(* IEC 61131-3 sources: HMITools/, 11 files *)

(* ---- GetDataObjectList.st ---- *)
(*  *)
FUNCTION GetDataObjectList

		//Keep track of the objects that we've gone through
	//unsigned int objectIndex = 0;
	objectIndex:= 0;

	//Number of variables that have been found
	numberVariables:=0;
	duplicate:=0;
	index:=0;

	//Check for valid inputs
	IF( List = 0 ) THEN
		GetDataObjectList:=0;
		RETURN;
	END_IF

	//Clear out any bad data
	Files ACCESS List;
	brsmemset(ADR(Files ),0,MaxObjects*(LIST_BOX_STRING_SIZE+1));

	//Look through all the objects
	WHILE( MO_list(objectIndex, ADR(objectIndex), ADR(Item)) = 0 AND numberVariables < MaxObjects)DO
		//If it is a cyclic object check if it has the variable
		duplicate:=0;
		IF( Item.type = 16#41) THEN
			FOR index:= 0 TO numberVariables DO
				IF(brsstrcmp(ADR(Item.name),ADR(Files[index]))=0)THEN
					duplicate:=1;
					EXIT;
				END_IF
			END_FOR
			IF(NOT duplicate) THEN
				brsstrcpy( ADR(Files[numberVariables]),ADR(Item.name));
				numberVariables:=numberVariables+1;
			END_IF
		END_IF
	END_WHILE

	//Return the number of found variables to make it easy to add to the list outside the function.
	GetDataObjectList:= numberVariables;

END_FUNCTION

(* ---- HMI_Lock.st ---- *)
(********************************************************************
 * COPYRIGHT --
 ********************************************************************
 * Library: HMI_Basic
 * File: HMI_Lock.st
 * Author: David
 * Created: May 03, 2011
 ********************************************************************
 * Implementation of library HMI_Basic
 ********************************************************************)

(****************************************************************)
(* Lock an item on the screen 									*)
(****************************************************************)

(* Function			DONE and TESTED DFB 20110503 *)

FUNCTION HMI_Lock

(****************************************************************)
(* Set return value to get rid of compiler error				*)
(****************************************************************)

HMI_Lock:=	FALSE;

(****************************************************************)
(* Set/clear proper bit in StatusDP								*)
(****************************************************************)

StatusDP.HMI_STATBIT_LOCK:=	HMI_LOCKED;

END_FUNCTION

(* ---- HMI_OpenTouchpad.st ---- *)
(********************************************************************
 * COPYRIGHT --
 ********************************************************************
 * Library: HMI_Basic
 * File: HMI_OpenTouchpad.st
 * Author: David
 * Created: May 04, 2011
 ********************************************************************
 * Implementation of library HMI_Basic
 ********************************************************************)

(********************************************************************)
(* Opens the touchpad for an item on the screen 					*)
(********************************************************************)

(* Function			DONE and TESTED DFB 20110504 *)

FUNCTION HMI_OpenTouchpad

(****************************************************************)
(* Set return value to get rid of compiler error				*)
(****************************************************************)

HMI_OpenTouchpad:=	FALSE;

(****************************************************************)
(* Set/clear proper bit in StatusDP								*)
(****************************************************************)

StatusDP.HMI_STATBIT_TOUCHPAD:=	1;

END_FUNCTION

(* ---- HMI_ResetFocus.st ---- *)
(********************************************************************
 * COPYRIGHT --
 ********************************************************************
 * Library: HMI_Basic
 * File: HMI_ResetFocus.st
 * Author: David
 * Created: May 04, 2011
 ********************************************************************
 * Implementation of library HMI_Basic
 ********************************************************************)

(************************************************************************************)
(* Resets the focus bit for an item on the screen. THIS DOES NOT MOVE THE FOCUS!	*)
(************************************************************************************)

(* Function			DONE and TESTED DFB 20110504 *)

FUNCTION HMI_ResetFocus

(****************************************************************)
(* Set return value to get rid of compiler error				*)
(****************************************************************)

HMI_ResetFocus:=	FALSE;

(****************************************************************)
(* Set/clear proper bit in StatusDP								*)
(****************************************************************)

StatusDP.HMI_STATBIT_FOCUS:=	0;

END_FUNCTION

(* ---- HMI_SetFocus.st ---- *)
(********************************************************************
 * COPYRIGHT --
 ********************************************************************
 * Library: HMI_Basic
 * File: HMI_SetFocus.st
 * Author: David
 * Created: May 04, 2011
 ********************************************************************
 * Implementation of library HMI_Basic
 ********************************************************************)

(********************************************************************)
(* Sets the focus for an item on the screen. FOCUS MUST BE RESET!	*)
(********************************************************************)

(* Function			DONE and TESTED DFB 20110504 *)

FUNCTION HMI_SetFocus

(****************************************************************)
(* Set return value to get rid of compiler error				*)
(****************************************************************)

HMI_SetFocus:=	FALSE;

(****************************************************************)
(* Set/clear proper bit in StatusDP								*)
(****************************************************************)

StatusDP.HMI_STATBIT_FOCUS:=	1;

END_FUNCTION

(* ---- HMI_Show.st ---- *)
(********************************************************************
 * COPYRIGHT --
 ********************************************************************
 * Library: HMI_Basic
 * File: HMI_Show.st
 * Author: David
 * Created: May 03, 2011
 ********************************************************************
 * Implementation of library HMI_Basic
 ********************************************************************)

(****************************************************************)
(* Show an item on the screen 									*)
(****************************************************************)

(* Function			DONE and TESTED DFB 20110503 *)

FUNCTION HMI_Show

(****************************************************************)
(* Set return value to get rid of compiler error				*)
(****************************************************************)

HMI_Show:=	FALSE;

(****************************************************************)
(* Set/clear proper bit in StatusDP								*)
(****************************************************************)

StatusDP.HMI_STATBIT_VIS:=	HMI_VISIBLE;

END_FUNCTION

(* ---- HMI_Unlock.st ---- *)
(********************************************************************
 * COPYRIGHT --
 ********************************************************************
 * Library: HMI_Basic
 * File: HMI_Unlock.st
 * Author: David
 * Created: May 03, 2011
 ********************************************************************
 * Implementation of library HMI_Basic
 ********************************************************************)

(****************************************************************)
(* Unlock an item on the screen 								*)
(****************************************************************)

(* Function			DONE and TESTED DFB 20110503 *)

FUNCTION HMI_Unlock

(****************************************************************)
(* Set return value to get rid of compiler error				*)
(****************************************************************)

HMI_Unlock:=	FALSE;

(****************************************************************)
(* Set/clear proper bit in StatusDP								*)
(****************************************************************)

StatusDP.HMI_STATBIT_LOCK:=	HMI_UNLOCKED;

END_FUNCTION

(* ---- DirectoryFub.st ---- *)
(********************************************************************
 * COPYRIGHT -- Automation Resources Group
 ********************************************************************
 * Program: FileManager
 * File: Directory.st
 * Author: Josh
 * Created: April 01, 2012
 ********************************************************************
 * Implementation of program FileManager
 ********************************************************************)

(*  *)
FUNCTION_BLOCK DirectoryFub

IF FileList = 0 OR Enable = 0 THEN
	Updating:=0;
	RETURN;
END_IF

Files ACCESS FileList;

	// Step through all states faster by looping 5 times
	FOR index:=0 TO 5 DO

		CASE State OF
			0:
				DirectoryRead.enable:=0;
				//CurrentFileIndex:=0; This variable is never used again.
				Updating:=1;
				State:=1;

			1:
				DirectoryOpen.enable := 	TRUE;
				DirectoryOpen.pDevice := 	ADR(FileDevice);
				DirectoryOpen.pName := 		pPath;
				DirectoryOpen();
				IF DirectoryOpen.status < ERR_FUB_ENABLE_FALSE THEN
					IF DirectoryOpen.status = ERR_OK THEN
						Ident :=			DirectoryOpen.ident;
						DirectoryOpen.enable:=	 FALSE;
						State:= 			State+1;
					ELSE
						status:= 			DirectoryOpen.status;
						State:=				10;
					END_IF;
				ELSE
					EXIT;
				END_IF;
				brsmemset(ADR(Files),0,MaxValues*(LIST_BOX_STRING_SIZE+1));
				ListFileIndex:=		0;
				status:=			ERR_FUB_BUSY;

			2:
				//read directory
				DirectoryRead.enable := 	TRUE;
				DirectoryRead.ident := 		Ident;
				DirectoryRead.pData := 		ADR(DirData);
				DirectoryRead.data_len := 	SIZEOF(DirData);
				DirectoryRead();
				IF DirectoryRead.status < ERR_FUB_ENABLE_FALSE THEN
					IF DirectoryRead.status = ERR_OK THEN
						DirectoryRead.enable := FALSE;
						State:= 			State+1;
					ELSIF DirectoryRead.status = fiERR_NO_MORE_ENTRIES THEN
						NumFiles:= 			ListFileIndex;
						status:=			ERR_OK;
						State:=				5;
					ELSE
						IF DirectoryRead.status = 20799 THEN
							status:= FileIoGetSysError();
						ELSE
							status:= DirectoryRead.status;
						END_IF;
						State:=				10;
					END_IF;
				ELSE
					EXIT;
				END_IF;

			3:
				brsstrcpy(ADR(TempString),ADR(DirData.Filename));
				iNameFilter:=NameFilter;
				//If file extension filter defined
				IF FileExt <> '' THEN
					brsmemset(ADR(TempExtension),0,SIZEOF(TempExtension));
					TempExtension:=	'.';
					brsstrcat(ADR(TempExtension),ADR(FileExt));
					//item is a File, files are filtered
					IF DirData.Mode = fiFILE THEN
						//compare just the selected extension from the file name + extension (e.g. compare ".csv" from "testing.csv")
						IF ( brsmemcmp((ADR(TempString)+(brsstrlen(ADR(TempString))-(brsstrlen(ADR(TempExtension)))))
							, ADR(TempExtension)
							, brsstrlen(ADR(TempExtension))) = 0) THEN

							//convert NameFilter to lowercase
							brsmemset(ADR(lcNameFilter),0,SIZEOF(lcNameFilter));
							FOR i:= 0 TO (SIZEOF(NameFilter) - 1) DO
								brsmemcpy(ADR(IsolatedChar),(ADR(NameFilter) + i),SIZEOF(USINT));
								IF IsolatedChar = 0 THEN// OR IsolatedChar = 46 THEN//if null or '.', dont convert file extension to lc
									EXIT;
								ELSIF IsolatedChar >=  65 AND IsolatedChar <=  90  THEN//Uppser case ascii
									brsmemset((ADR(lcNameFilter) + i),(IsolatedChar + 32),SIZEOF(USINT));
								ELSE//lower case ascii
									brsmemset((ADR(lcNameFilter) + i),IsolatedChar,SIZEOF(USINT));
								END_IF;
							END_FOR;
							//convert TempString to lowercase
							brsmemset(ADR(lcTempString),0,SIZEOF(lcTempString));
							FOR i:= 0 TO (SIZEOF(TempString) - 1) DO
								brsmemcpy(ADR(IsolatedChar),(ADR(TempString) + i),SIZEOF(USINT));
								IF IsolatedChar = 0 THEN// OR IsolatedChar = 46 THEN//if null or '.', dont convert file extension to lc
									EXIT;
								ELSIF IsolatedChar >=  65 AND IsolatedChar <=  90  THEN//Uppser case ascii
									brsmemset((ADR(lcTempString) + i),(IsolatedChar + 32),SIZEOF(USINT));
								ELSE//lower case ascii
									brsmemset((ADR(lcTempString) + i),IsolatedChar,SIZEOF(USINT));
								END_IF;
							END_FOR;
							brsmemcpy(ADR(IsolatedChar),ADR(TempString),SIZEOF(USINT));

							//Compare both lower case strings
							//Check for hidden files
							IF (FIND(lcTempString, lcNameFilter) <> 0) AND (ShowHiddenFiles OR IsolatedChar <> 46) THEN
								brsstrcpy(ADR(Files[ListFileIndex]),ADR(DirData.Filename));
								ListFileIndex:=		ListFileIndex+1;
								State:= 			State+1;
							ELSE
								State:= 			State+1;
							END_IF;

						ELSE
							State:= 			State+1;
						END_IF
					//item is a Directory, directories are not filtered
					ELSIF EnableDirectorySearch AND (brsstrcmp(ADR(DirData.Filename),ADR('.')) <> 0) THEN
						IF ((brsstrcmp(pPath,ADR('')) = 0) AND ((brsstrcmp(ADR(DirData.Filename),ADR('..')) = 0))) THEN
							State:=				State+1;
						ELSE
							brsstrcpy(ADR(Files[ListFileIndex]),ADR('\'));
							brsstrcat(ADR(Files[ListFileIndex]),ADR(DirData.Filename));
							ListFileIndex:=		ListFileIndex+1;
							State:=				State+1;
						END_IF;
					ELSE//if a directory and enabledirectorysearch is false
						State:= 				State+1;
					END_IF;
				//No extension filter defined
				ELSE
					//item is a File, files are filtered
					IF DirData.Mode = fiFILE THEN
						//convert NameFilter to lowercase
						brsmemset(ADR(lcNameFilter),0,SIZEOF(lcNameFilter));
						FOR i:= 0 TO (SIZEOF(NameFilter) - 1) DO
							brsmemcpy(ADR(IsolatedChar),(ADR(NameFilter) + i),SIZEOF(USINT));
							IF IsolatedChar = 0 THEN// OR IsolatedChar = 46 THEN//if null or '.', dont convert file extension to lc
								EXIT;
							ELSIF IsolatedChar >=  65 AND IsolatedChar <=  90  THEN//Uppser case ascii
								brsmemset((ADR(lcNameFilter) + i),(IsolatedChar + 32),SIZEOF(USINT));
							ELSE//lower case ascii
								brsmemset((ADR(lcNameFilter) + i),IsolatedChar,SIZEOF(USINT));
							END_IF;
						END_FOR;
						//convert TempString to lowercase
						brsmemset(ADR(lcTempString),0,SIZEOF(lcTempString));
						FOR i:= 0 TO (SIZEOF(TempString) - 1) DO
							brsmemcpy(ADR(IsolatedChar),(ADR(TempString) + i),SIZEOF(USINT));
							IF IsolatedChar = 0 THEN//OR IsolatedChar = 46 THEN//if null or '.', dont convert file extension to lc
								EXIT;
							ELSIF IsolatedChar >=  65 AND IsolatedChar <=  90  THEN//Uppser case ascii
								brsmemset((ADR(lcTempString) + i),(IsolatedChar + 32),SIZEOF(USINT));
							ELSE//lower case ascii
								brsmemset((ADR(lcTempString) + i),IsolatedChar,SIZEOF(USINT));
							END_IF;
						END_FOR;

						brsmemcpy(ADR(IsolatedChar),ADR(TempString),SIZEOF(USINT));

						//Compare both lower case strings
						//Check for hidden files
						IF (FIND(lcTempString, lcNameFilter) <> 0) AND (ShowHiddenFiles OR IsolatedChar <> 46) THEN
							brsstrcpy(ADR(Files[ListFileIndex]),ADR(DirData.Filename));
							ListFileIndex:=		ListFileIndex+1;
							State:= 			State+1;
						ELSE
							State:= 			State+1;
						END_IF;

					//item is a Directory, directories are not filtered
					ELSIF EnableDirectorySearch AND (brsstrcmp(ADR(DirData.Filename),ADR('.')) <> 0) THEN //item is a Directory, directories are not filtered
						IF ((brsstrcmp(pPath,ADR('')) = 0) AND ((brsstrcmp(ADR(DirData.Filename),ADR('..')) = 0))) THEN
							State:=				State+1;
						ELSE
							brsstrcpy(ADR(Files[ListFileIndex]),ADR('\'));
							brsstrcat(ADR(Files[ListFileIndex]),ADR(DirData.Filename));
							ListFileIndex:=		ListFileIndex+1;
							State:=				State+1;
						END_IF;
					ELSE//if a directory and enabledirectorysearch is false
						State:= 				State+1;
					END_IF;
				END_IF;

			4:
				IF ListFileIndex = MaxValues THEN
					status:=	ERR_OK;
					NumFiles:= 	ListFileIndex;
					State:=		5;
				ELSE
					State:=		2;
				END_IF;

			5:
				DirectoryClose.enable := 	TRUE;
				DirectoryClose.ident := 	Ident;
				DirectoryClose();
				IF DirectoryClose.status = ERR_OK THEN
					DirectoryClose.enable := FALSE;
					State:= 				6;
				END_IF;

			10:
				Initialized:=	1;
				UpdateTimer.IN:=1;
				IF UpdateTimer.Q OR iNameFilter<>NameFilter OR Refresh THEN
					Refresh:= 	0;
					State:=		0;
				END_IF

			ELSE
				Initialized:=	1;
				Updating:=		0;
				UpdateTimer.IN:=1;
				IF UpdateTimer.Q OR iNameFilter<>NameFilter OR Refresh THEN
					Refresh:= 	0;
					State:=		0;
				END_IF
		END_CASE;
	END_FOR;

UpdateTimer.PT:=T#60s;
UpdateTimer();
UpdateTimer.IN:=0;

END_FUNCTION_BLOCK

(* ---- HMI_File_Browse.st ---- *)
(********************************************************************
 * COPYRIGHT --
 ********************************************************************
 * Library: HMITools
 * File: HMIFileBrowse.st
 * Author: Josh
 * Created: November 08, 2012
 ********************************************************************
 * Implementation of library HMITools
 ********************************************************************)

FUNCTION_BLOCK HMIFileBrowse
	// Error Checks

	IF pFileList = 0 THEN
		Status :=	'Invalid entry: FileList = 0';
		RETURN;
	END_IF;

	IF MaxFiles = 0 THEN
		Status :=	'Invalid entry: MaxFiles = 0';
		RETURN;
	END_IF;

	IF pFileExtList = 0
		AND MaxExt <> 0 THEN
		Status :=	'Invalid entry: pFileExtList = 0';
		RETURN;
	END_IF;

	IF pFileExtList <> 0
		AND MaxExt = 0 THEN
		Status :=	'Invalid entry: MaxExt = 0';
		RETURN;
	END_IF;

	IF FileDevice = '' THEN
		Status :=	'Invalid entry: FileDevice = 0';
		RETURN;
	END_IF;

	IF BrowseToDirectory AND EnableDirectorySearch = FALSE THEN
		BrowseToDirectory:=	FALSE;
		Status :=	'Please enable directory search';
	END_IF;

	IF Internal.TempFileList = 0 THEN
		TMP_alloc(SIZEOF(FileSelection) * MaxFiles ,ADR(Internal.TempFileList));
	END_IF

	Internal.FileExtensionSelector.IndexDP:=FileExtIndex;
	Internal.FileExtensionSelector.Enable:=Enable;
	Internal.FileExtensionSelector.MaxDP:=MaxExt;
	Internal.FileExtensionSelector.Selection:=ADR(FileExtSelection);
	IF pFileExtList <> 0 THEN
		Internal.FileExtensionSelector.SelectionList:=pFileExtList;
	END_IF;
	Internal.FileExtensionSelector();

	Internal.Directory.Enable:=		Enable AND NOT EnableDataObjects;
	Internal.Directory.MaxValues:= 	MaxFiles;
	IF Internal.TempFileList <> 0 THEN
		Internal.Directory.FileList:=Internal.TempFileList;
	ELSE
		Internal.Directory.FileList:=pFileList;
	END_IF

	//If initial path given
	IF pDirectorySearchPath <> 0
		AND Internal.InternalBrowsingPath = '' THEN
		brsstrcpy(ADR(CurrentPath),pDirectorySearchPath);
	END_IF;

	//if command to add FileSelection to browsing path,
	IF BrowseToDirectory
		AND FileSelection <> '\..'
		AND FileSelection <> '' THEN
		BrowseToDirectory := 	FALSE;
		Refresh := 1; // do an update and navigate to directory

		//Running directory path check
		brsmemcpy(ADR(Internal.IsolatedChar),ADR(FileSelection),SIZEOF(USINT));
		IF Internal.IsolatedChar = ASCII_BACKSLASH THEN
			//add selected file to internal path
			brsstrcat(ADR(Internal.InternalBrowsingPath),(ADR(FileSelection) + 1));//Don't add first character "\" to the browsing path
			brsstrcat(ADR(Internal.InternalBrowsingPath),ADR('\'));
			//reset current path
			brsmemset(ADR(CurrentPath),0,SIZEOF(CurrentPath));
			//repopulate current path with directory path input
			IF pDirectorySearchPath <> 0 THEN
				brsstrcpy(ADR(CurrentPath),(pDirectorySearchPath));
			END_IF;
			brsstrcat(ADR(CurrentPath),ADR(Internal.InternalBrowsingPath));
			//RESET FileSelection
			FileIndex:=				-1;
			FileSelection:=			'';
		ELSE
			Status:= 				'Invalid Internal.Directory';
		END_IF;
	//If command GoToParentInternal.Directory
	ELSIF BrowseToDirectory AND FileSelection = '\..' THEN
		BrowseToDirectory :=	FALSE;
		Refresh := 1; // do an update and navigate to directory
		Internal.PathStrSize:=		UDINT_TO_UINT(brsstrlen(ADR(Internal.InternalBrowsingPath)));
		IF Internal.InternalBrowsingPath = '' THEN//at highest allowed directory, indicated by input FileDevice and Path
			Status:= 				'Invalid Internal.Directory';
		ELSE
			brsmemset(ADR(Internal.InternalBrowsingPath) +(Internal.PathStrSize - 1 ),0,SIZEOF(USINT));//remove the last character "\"
			FOR Internal.i:= 1 TO Internal.PathStrSize DO
				//isolate a single character off of the path string
				brsmemcpy(ADR(Internal.IsolatedChar),ADR(Internal.InternalBrowsingPath)+(Internal.PathStrSize-Internal.i),SIZEOF(USINT));
				//if no characters left
				IF brsstrcmp(ADR(Internal.InternalBrowsingPath),ADR('')) = 0 THEN
					EXIT;
				//if found a backslash character at the end of the string, remove it and exit
				ELSIF Internal.IsolatedChar = ASCII_BACKSLASH  THEN
					EXIT;
				//else it's a normal character, remove it
				ELSE
					brsmemset(ADR(Internal.InternalBrowsingPath) +(Internal.PathStrSize-Internal.i),0,SIZEOF(USINT));
				END_IF;
			END_FOR;
		END_IF;
		//RESET FileSelection
		FileIndex:=		-1;
		FileSelection:=	'';
		//set output to current path
		brsmemset(ADR(CurrentPath),0,SIZEOF(CurrentPath));
		IF pDirectorySearchPath <> 0 THEN
			brsstrcpy(ADR(CurrentPath),pDirectorySearchPath);
		END_IF;
		brsstrcat(ADR(CurrentPath),ADR(Internal.InternalBrowsingPath));
	ELSIF BrowseToDirectory AND FileSelection = '' THEN
		BrowseToDirectory :=	FALSE;
		Status :=	'Invalid Internal.Directory';
	END_IF;

	//If selecting a file from listbox don't update name filter
	IF FileIndex < 0 THEN
		Internal.NameFilter :=	FileSelection;
	END_IF

	//temporarly display the filter being applied
	IF FileIndex < 0 AND Internal.NameFilter <> '' THEN
		Status :=		'Filter "';
		brsstrcat(ADR(Status),ADR(Internal.NameFilter));
		brsstrcat(ADR(Status),ADR('" applied'));
	END_IF

	//Reset Internal.NameFilter if a space character is the first character
	IF (brsmemcmp(ADR(FileSelection),ADR(' '),1) = 0) THEN
		Internal.NameFilter:=		'';
		FileSelection :=	'';
		Status :=			'Name filter removed';
	END_IF

	Internal.Directory.FileExt:=		FileExtSelection;
	Internal.Directory.FileDevice:=		FileDevice;
	Internal.Directory.EnableDirectorySearch:=	EnableDirectorySearch;
	Internal.Directory.pPath:=			ADR(CurrentPath);
	Internal.Directory.NameFilter:= 	Internal.NameFilter;

	IF (Refresh) THEN
		Internal.Directory.Refresh := 1;
	END_IF

	Internal.Directory();
	Refresh := 0;

	IF EnableDataObjects AND Enable THEN
		NumFiles:= GetDataObjectList(Internal.Directory.FileList,MaxFiles);
	ELSE
		NumFiles:= 				Internal.Directory.NumFiles;
	END_IF

	IF NOT Internal.Directory.Updating
		AND Internal.TempFileList <> 0
		AND Enable
		THEN
		brsmemcpy(pFileList,Internal.TempFileList,Internal.Directory.MaxValues*(LIST_BOX_STRING_SIZE+1));
	END_IF

	//If manually changing FileSelection, reset with FileIndex to update the Internal.NameFilter
	IF Internal.oldFileSelection <> FileSelection AND FileIndex = Internal.oldFileIndex THEN
		FileIndex:=	-1;
	END_IF;

	Internal.TempFileSelection := FileSelection;

	Internal.FileNameSelector.IndexDP:=		FileIndex;
	Internal.FileNameSelector.Enable:=		Enable;
	Internal.FileNameSelector.Enable:=		TRUE;
	Internal.FileNameSelector.MaxDP:=		Internal.Directory.NumFiles;
	Internal.FileNameSelector.Selection:=	ADR(Internal.TempFileSelection);
	Internal.FileNameSelector.SelectionList:=	pFileList;
	Internal.FileNameSelector();

	//We need to read back the found index to ensure that we aren't constantly updating
	FileIndex:= Internal.FileNameSelector.IndexDP;

	FileExtIndex:=	Internal.FileExtensionSelector.IndexDP;
	//FileIndex:=Internal.oldFileSelection.IndexDP;

	IF FileIndex > -1 THEN
		FileSelection:=		Internal.TempFileSelection;
		Internal.oldFileSelection:=	FileSelection;
	END_IF;

	CompletionDP:=Internal.FileNameSelector.CompletionDP;

	//If manually changing FileSelection, reset with FileIndex to update the Internal.NameFilter
	IF Internal.oldFileSelection <> FileSelection AND FileIndex = Internal.oldFileIndex THEN
		FileIndex:=	-1;
		Internal.oldFileSelection:=	FileSelection;
	ELSE
		Internal.oldFileSelection:=	FileSelection;
	END_IF;
	IF Internal.oldFileIndex <> FileIndex THEN
		Internal.oldFileIndex:=		FileIndex;
	END_IF;

	//Reset Error String Handling
	IF Status <> '' THEN
		Internal.TON_0.IN := 	TRUE;
		Internal.TON_0.PT := 	T#2s;
		IF Internal.TON_0.Q THEN
			Internal.TON_0.IN:=	FALSE;
			brsmemset(ADR(Status),0,SIZEOF(Status));
		END_IF;
	ELSE
		Internal.TON_0.IN := 	FALSE;
	END_IF;
	Internal.TON_0();

	//If no files or directories found
	IF NumFiles = 0 AND EnableDirectorySearch = FALSE THEN
		Status:=	'No files found';
	ELSIF NumFiles = 0 AND EnableDirectorySearch = TRUE THEN
		Status:=	'No items found';
	END_IF;

END_FUNCTION_BLOCK

(* ---- Trend_ZoomScroll.st ---- *)
(********************************************************************
 * COPYRIGHT -- Automation Resources Group
 ********************************************************************
 * Library: HMITools
 * File: Trend_ZoomScroll.st
 * Author: David
 * Created: October 25, 2010
 ********************************************************************
 * Implementation of library HMITools
 ********************************************************************)

(********************************************************************)
(* Smart handling of trend zooming and scaling 						*)
(********************************************************************)

(* Functionality			DONE and TESTED DFB *)

FUNCTION_BLOCK Trend_ZoomScroll

	(* Initialize values on startup *)

	IF( NOT(Init) )THEN

 		Init:=	1;
		Reset:=	1;

	END_IF

	(* Reset *)

	IF( Reset )THEN

 		Reset:=		0;

		ZoomDP:=	1;
		ScrollDP:=	0;
		ModeDP:=	1;

	END_IF

	(* Zoom *)

	(* Check ZoomBase *)

	IF( ZoomBase < 1 )THEN

		(* If ZoomBase is less than 1, this will cause problems.
			Default to a ZoomBase of 1. This cancels out all Zooming *)

 		ZoomBase:=	1;

	END_IF

	IF( ZoomIn )THEN

 		ZoomIn:=	0;

		Midpt:=		ScrollDP + (0.5 / ZoomDP);	(* Midpt is ScrollDP (StartPt_curr) + Range_curr/2; Range_curr is 1/ZoomDP_curr *)
		ZoomDP:=	ZoomDP * ZoomBase; 			(* Zoom is increased by ZoomBase *)
		ScrollDP:=	Midpt - (0.5 / ZoomDP);		(* New Scroll is Midpt - Range_new/2; Range_new is 1/ZoomDP_new *)

	END_IF

	IF( ZoomOut )THEN

 		ZoomOut:=	0;

		Midpt:=		ScrollDP + (0.5 / ZoomDP);	(* Midpt is ScrollDP (StartPt_curr) + Range_curr/2; Range_curr is 1/ZoomDP_curr *)
		ZoomDP:=	ZoomDP / ZoomBase; 			(* Zoom is decreased by ZoomBase *)
		ScrollDP:=	Midpt - (0.5 / ZoomDP);		(* New Scroll is Midpt - Range_new/2; Range_new is 1/ZoomDP_new *)

	END_IF

	(* Scroll *)

	(* Check ScrollBase *)

	IF( ScrollBase < 0 )THEN

		(* If ScrollBase is less than 0, this will cause problems.
			Default to a ScrollBase of 0. This cancels out all Scrolling *)

 		ScrollBase:=	0;

	END_IF

	IF( ScrollNeg )THEN

 		ScrollNeg:=	0;

		ScrollDP:=	ScrollDP - ScrollBase / ZoomDP;	(* Decrease ScrollDP by percentage (ScrollBase) of Range. Range is 1/ZoomDP *)

	END_IF

	IF( ScrollPos )THEN

 		ScrollPos:=	0;

		ScrollDP:=	ScrollDP + ScrollBase / ZoomDP; (* Increase ScrollDP by percentage (ScrollBase) of Range. Range is 1/ZoomDP *)

	END_IF

END_FUNCTION_BLOCK

(* ---- UpdateFiles.st ---- *)
(********************************************************************
 * COPYRIGHT --
 ********************************************************************
 * Program: RecipeUpdater
 * File: UpdateFiles.st
 * Author: Josh
 * Created: June 17, 2015
 ********************************************************************
 * Implementation of program RecipeUpdater
 ********************************************************************)

(* TODO: Add your comment here *)
FUNCTION_BLOCK FileQueue

	CASE internal.State OF

		RecipeUpdater_ST_IDLE:
			Busy := FALSE;
			IF Next THEN
				Busy:=	TRUE;
				internal.DirRead.entry:= 0;
				internal.State:= RecipeUpdater_ST_ReadDirectory;
			END_IF

		RecipeUpdater_ST_ReadDirectory:

			IF internal.DirRead.status = 0 THEN
				internal.DirRead.enable:= FALSE;
				IF internal.CurrentFile.Filename[0] <> 46 THEN
					internal.State:= RecipeUpdater_ST_ReadFile;
					brsstrcpy(ADR(FileName),ADR(internal.CurrentFile.Filename));
				ELSE
					internal.DirRead.entry:= internal.DirRead.entry+1;
				END_IF
			ELSIF internal.DirRead.status = ERR_FUB_BUSY
				OR internal.DirRead.status = ERR_FUB_ENABLE_FALSE
				THEN
				internal.DirRead.enable:= TRUE;
			ELSIF internal.DirRead.status = fiERR_NO_MORE_ENTRIES
				THEN
				internal.State:= RecipeUpdater_ST_Done;
			ELSE
				Error:=	TRUE;
				ErrorID:=	internal.DirRead.status;
				internal.State:= RecipeUpdater_ST_Done;
			END_IF

		RecipeUpdater_ST_ReadFile:

			Execute:=	TRUE;
			IF NOT Next THEN
				Execute:=	FALSE;
				internal.State:= RecipeUpdater_ST_WAIT;
			ELSIF Cancel THEN
				Execute:=	FALSE;
				internal.State:= RecipeUpdater_ST_Done;
			END_IF

		RecipeUpdater_ST_WAIT:

			Execute:=	FALSE;
			IF Next THEN
				internal.State:= RecipeUpdater_ST_ReadDirectory;
				internal.DirRead.entry:= internal.DirRead.entry+1;
			ELSIF Cancel THEN
				Execute:=	FALSE;
				internal.State:= RecipeUpdater_ST_Done;
			END_IF

		RecipeUpdater_ST_Done:

			Done:= TRUE;
			Busy:=0;

			IF NOT Next
				AND NOT Cancel
				THEN
				Error:=0;
				Done:=0;
				ErrorID:=0;
				internal.State:= RecipeUpdater_ST_IDLE;
			END_IF

		RecipeUpdater_ST_:

	END_CASE

	internal.DirRead.option:=	fiFILE;
	internal.DirRead.pData:=	ADR(internal.CurrentFile);
	internal.DirRead.data_len:= SIZEOF(internal.CurrentFile);
	internal.DirRead.pDevice:=	ADR(FileDevice);
	internal.DirRead.pPath:=	ADR(Path);
	internal.DirRead();
	internal.DirRead.enable:= FALSE;

END_FUNCTION_BLOCK
